// TIA Portal V17 export
// export: Created 2024-08-07T21:43:59.0989886Z, ExportSetting WithDefaults, DisplayName Totally Integrated Automation Portal, DisplayVersion V17 Update 7, DisplayName TIA Portal Openness, DisplayVersion V17 Update 7, DisplayName TIA Portal Version Control Interface, DisplayVersion V17, DisplayName SINAMICS Startdrive Advanced, DisplayVersion V17 SP2, DisplayName SINAMICS Startdrive G110M, G120, G120C, G120D, G120P, G115D, DisplayVersion V17 SP2, DisplayName SINAMICS Startdrive G130, G150, S120, S150, SINAMICS MV, S210, DisplayVersion V17 SP2, DisplayName STEP 7 Professional, DisplayVersion V17 Update 7, DisplayName STEP 7 Safety, DisplayVersion V17 Update 6, DisplayName WinCC Advanced / Unified PC, DisplayVersion V17 Update 7
FUNCTION_BLOCK "FB_DTM"   // FB301, LAD
{ S7_Optimized_Access := 'TRUE' }
VERSION : 0.1
// stored: AutoNumber false, IsIECCheckEnabled false, IsRetainMemResEnabled false, MemoryReserve 100, SetENOAutomatically false, UDAEnableTagReadback false
   VAR_INPUT
      Req : Bool;
      TriggerReady : Bool;
      TriggerAck : Bool;
      ResultsAvailable : Bool;
      ResultID : Word;
      ResultCode : Word;
      ResultLenght : Word;
      ResultData : "udt_DTM_resultData";
   END_VAR
   VAR_OUTPUT
      TriggerEnable : Bool;
      Trigger : Bool;
      ResultsAck : Bool;
      DataStr : String;
   END_VAR
   VAR
      ResultPending { ExternalAccessible := 'False'; ExternalVisible := 'False'; ExternalWritable := 'False'} : Bool;
      LatestResults { ExternalAccessible := 'False'; ExternalVisible := 'False'; ExternalWritable := 'False'} : Struct
         ID { ExternalAccessible := 'False'; ExternalVisible := 'False'; ExternalWritable := 'False'} : Int;
         Flags { ExternalAccessible := 'False'; ExternalVisible := 'False'; ExternalWritable := 'False'} : Int;
         Length { ExternalAccessible := 'False'; ExternalVisible := 'False'; ExternalWritable := 'False'} : Int;
         Value { ExternalAccessible := 'False'; ExternalVisible := 'False'; ExternalWritable := 'False'} : Array[0..63] of Byte;
      END_STRUCT;
   END_VAR
   VAR CONSTANT
      test : Bool := true;
   END_VAR
   VAR_TEMP   // added for the SCL form of the ladder/FBD networks
      _w1 : Bool;
   END_VAR
BEGIN

REGION Network 1: DataMan Acquisition Control Module
   // Make sure triggering is enabled
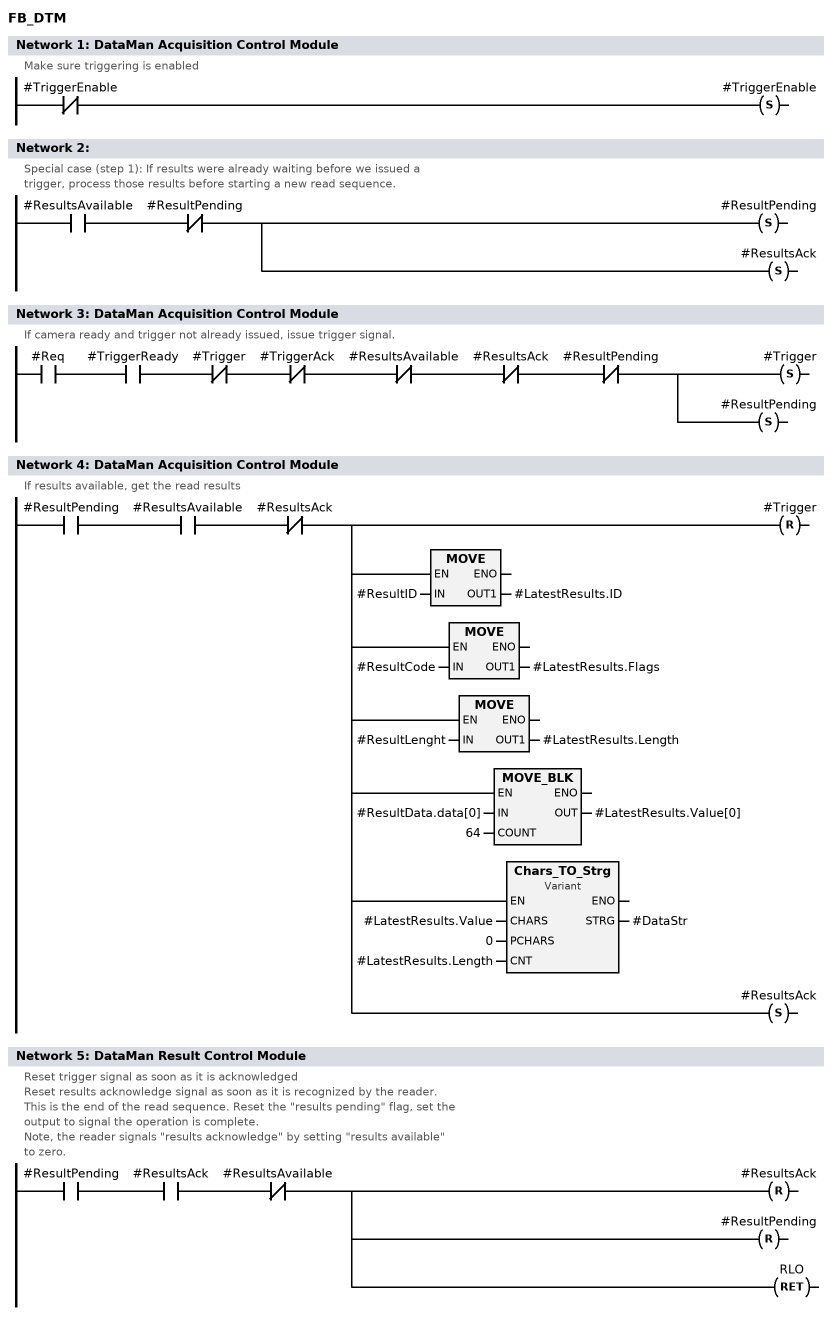
   RUNG wire#powerrail
      I_Contact( #TriggerEnable )
      S_Coil( #TriggerEnable )
   END_RUNG
   // the same network as SCL:
   IF NOT #TriggerEnable THEN #TriggerEnable := TRUE; END_IF;
END_REGION

REGION Network 2
   // Special case (step 1): If results were already waiting before we issued a 
   // trigger, process those results before starting a new read sequence.
   RUNG wire#powerrail
      Contact( #ResultsAvailable )
      I_Contact( #ResultPending )
      wire#w1
      S_Coil( #ResultPending )
   END_RUNG
   RUNG wire#w1
      S_Coil( #ResultsAck )
   END_RUNG
   // the same network as SCL:
   #_w1 := #ResultsAvailable AND NOT #ResultPending;
   IF #_w1 THEN
       #ResultPending := TRUE;
       #ResultsAck := TRUE;
   END_IF;
END_REGION

REGION Network 3: DataMan Acquisition Control Module
   // If camera ready and trigger not already issued, issue trigger signal.
   RUNG wire#powerrail
      Contact( #Req )
      Contact( #TriggerReady )
      I_Contact( #Trigger )
      I_Contact( #TriggerAck )
      I_Contact( #ResultsAvailable )
      I_Contact( #ResultsAck )
      I_Contact( #ResultPending )
      wire#w1
      S_Coil( #Trigger )
   END_RUNG
   RUNG wire#w1
      S_Coil( #ResultPending )
   END_RUNG
   // the same network as SCL:
   #_w1 := #Req AND #TriggerReady AND NOT #Trigger AND NOT #TriggerAck AND NOT #ResultsAvailable AND NOT #ResultsAck AND NOT #ResultPending;
   IF #_w1 THEN
       #Trigger := TRUE;
       #ResultPending := TRUE;
   END_IF;
END_REGION

REGION Network 4: DataMan Acquisition Control Module
   // If results available, get the read results
   IF #ResultPending AND #ResultsAvailable AND NOT #ResultsAck THEN
       #Trigger := FALSE;
       #LatestResults.ID := #ResultID;
       #LatestResults.Flags := #ResultCode;
       #LatestResults.Length := #ResultLenght;
       MOVE_BLK(IN := #ResultData.data[0], COUNT := 64, OUT => #LatestResults.Value[0]);
       Chars_TO_Strg(Chars := #LatestResults.Value, pChars := 0, Cnt := #LatestResults.Length, Strg => #DataStr);
       #ResultsAck := TRUE;
   END_IF;
END_REGION

REGION Network 5: DataMan Result Control Module
   // Reset trigger signal as soon as it is acknowledged 
   // Reset results acknowledge signal as soon as it is recognized by the reader.
   // 
   // This is the end of the read sequence. Reset the "results pending" flag, set the 
   // output to signal the operation is complete.
   // 
   // Note, the reader signals "results acknowledge" by setting "results available" 
   // to zero.
   #_w1 := #ResultPending AND #ResultsAck AND NOT #ResultsAvailable;
   IF #_w1 THEN
       #ResultsAck := FALSE;
       #ResultPending := FALSE;
       ENO := TRUE;
       RETURN;
   END_IF;
END_REGION
END_FUNCTION_BLOCK
